{attribute 'GeneratedUsingTerminal: EK1100-0000-0018'}
{attribute addProperty BoxType "EK1100-0000-0018"}
{attribute addProperty Id "Term_15_EL3403EL3403_812980A665Term_16_EK1122Term_16_EK1122_50B0E770140Term_23_EL3024EL3024_C6E76B5A40"}
{attribute addProperty CRC "646938495"}
{attribute addProperty Size "245"}
TYPE Term_14_EK1100_268F7F7F EXTENDS EK1100_1FC0878B :
STRUCT
	{attribute addProperty Name "Term_15_EL3403"}
	{attribute addProperty PreviousPort "Term 14 (EK1100) : B"}
	Term_15_EL3403 : EL3403_812980A6;
	{attribute addProperty Name "Term_16_EK1122"}
	{attribute addProperty PreviousPort "Term 15 (EL3403) : B"}
	Term_16_EK1122 : Term_16_EK1122_50B0E770;
	{attribute addProperty Name "Term_23_EL3024"}
	{attribute addProperty PreviousPort "Term 16 (EK1122) : C"}
	Term_23_EL3024 : EL3024_C6E76B5A;
END_STRUCT
END_TYPE

(* stored: Version 1.2.0.0, ProductVersion 3.1.4024.9
   DUT Term_14_EK1100_268F7F7F: Id {fbf61aeb-d2e9-0f45-236a-1eb7441d809e} *)
